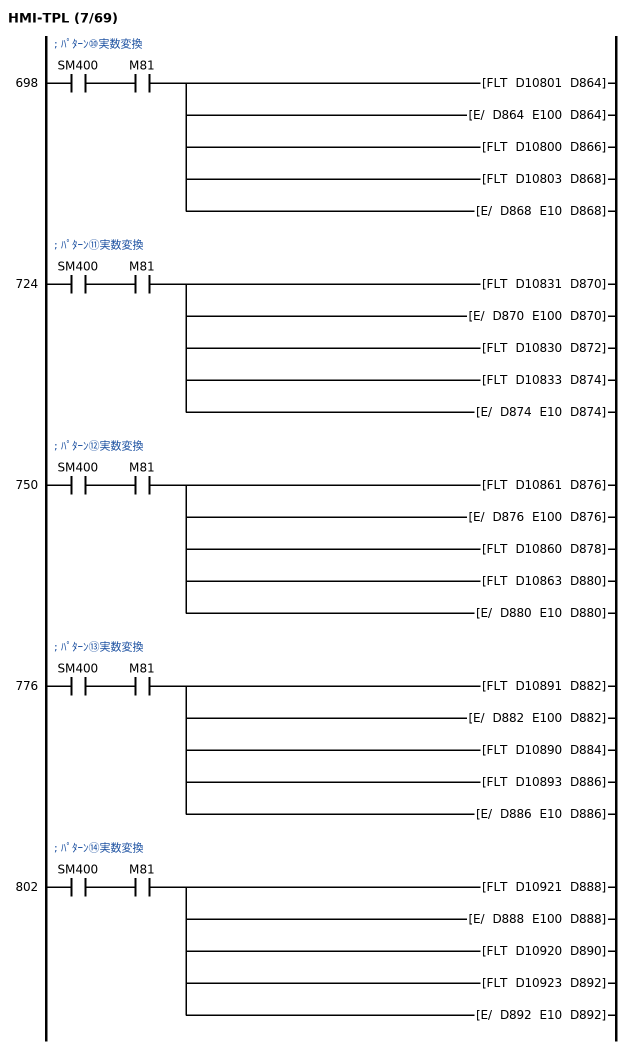
[picture p408: ladder of HMI-TPL, rungs at steps 698 to 802]
; ﾊﾟﾀｰﾝ⑩実数変換
698   LD      SM400
      AND     M81
      FLT     D10801 D864
      E/      D864 E100 D864
      FLT     D10800 D866
      FLT     D10803 D868
      E/      D868 E10 D868
; ﾊﾟﾀｰﾝ⑪実数変換
724   LD      SM400
      AND     M81
      FLT     D10831 D870
      E/      D870 E100 D870
      FLT     D10830 D872
      FLT     D10833 D874
      E/      D874 E10 D874
; ﾊﾟﾀｰﾝ⑫実数変換
750   LD      SM400
      AND     M81
      FLT     D10861 D876
      E/      D876 E100 D876
      FLT     D10860 D878
      FLT     D10863 D880
      E/      D880 E10 D880
; ﾊﾟﾀｰﾝ⑬実数変換
776   LD      SM400
      AND     M81
      FLT     D10891 D882
      E/      D882 E100 D882
      FLT     D10890 D884
      FLT     D10893 D886
      E/      D886 E10 D886
; ﾊﾟﾀｰﾝ⑭実数変換
802   LD      SM400
      AND     M81
      FLT     D10921 D888
      E/      D888 E100 D888
      FLT     D10920 D890
      FLT     D10923 D892
      E/      D892 E10 D892
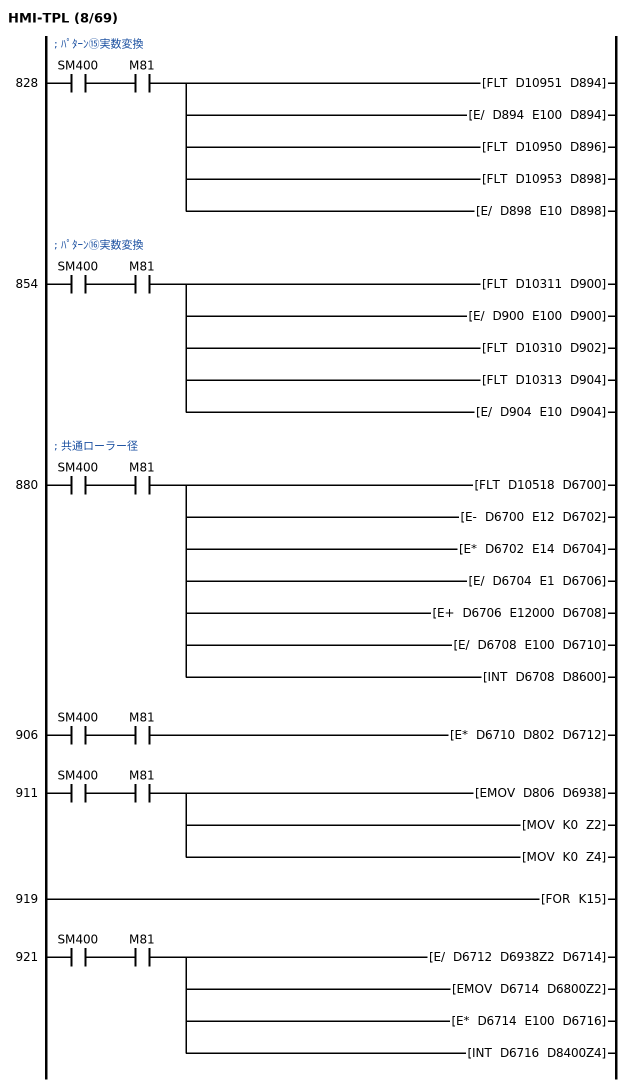
; ﾊﾟﾀｰﾝ⑮実数変換
828   LD      SM400
      AND     M81
      FLT     D10951 D894
      E/      D894 E100 D894
      FLT     D10950 D896
      FLT     D10953 D898
      E/      D898 E10 D898
; ﾊﾟﾀｰﾝ⑯実数変換
854   LD      SM400
      AND     M81
      FLT     D10311 D900
      E/      D900 E100 D900
      FLT     D10310 D902
      FLT     D10313 D904
      E/      D904 E10 D904
; 共通ローラー径
880   LD      SM400
      AND     M81
      FLT     D10518 D6700
      E-      D6700 E12 D6702
      E*      D6702 E14 D6704
      E/      D6704 E1 D6706
      E+      D6706 E12000 D6708
      E/      D6708 E100 D6710
      INT     D6708 D8600
906   LD      SM400
      AND     M81
      E*      D6710 D802 D6712
911   LD      SM400
      AND     M81
      EMOV    D806 D6938
      MOV     K0 Z2
      MOV     K0 Z4
919   FOR     K15
921   LD      SM400
      AND     M81
      E/      D6712 D6938Z2 D6714
      EMOV    D6714 D6800Z2
      E*      D6714 E100 D6716
      INT     D6716 D8400Z4
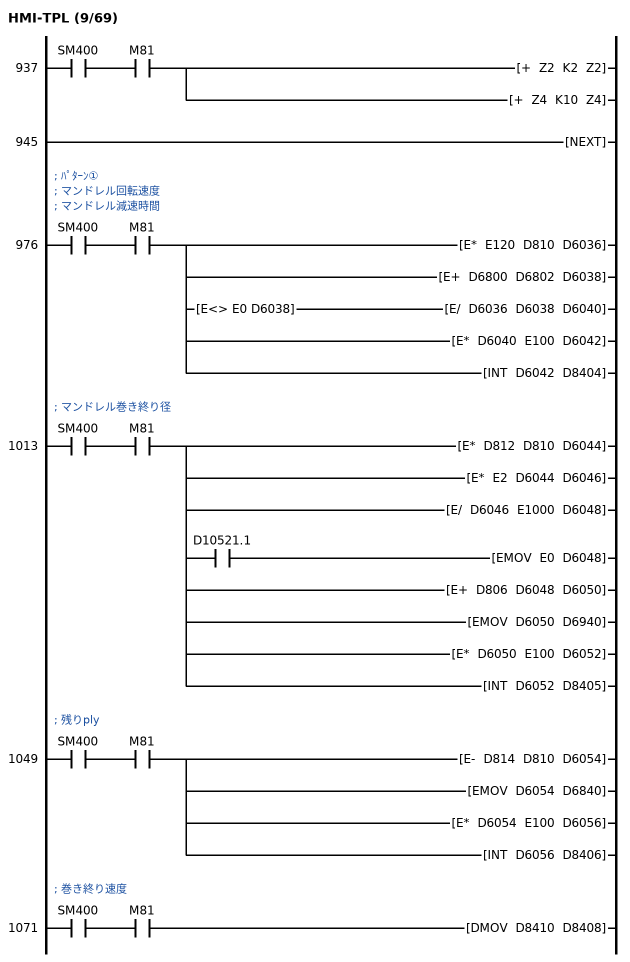
937   LD      SM400
      AND     M81
      +       Z2 K2 Z2
      +       Z4 K10 Z4
945   NEXT
; ﾊﾟﾀｰﾝ①
; マンドレル回転速度
; マンドレル減速時間
976   LD      SM400
      AND     M81
      E*      E120 D810 D6036
      E+      D6800 D6802 D6038
      MPS
      ANDE<>  E0 D6038
      E/      D6036 D6038 D6040
      MPP
      E*      D6040 E100 D6042
      INT     D6042 D8404
; マンドレル巻き終り径
1013  LD      SM400
      AND     M81
      E*      D812 D810 D6044
      E*      E2 D6044 D6046
      E/      D6046 E1000 D6048
      MPS
      AND     D10521.1
      EMOV    E0 D6048
      MPP
      E+      D806 D6048 D6050
      EMOV    D6050 D6940
      E*      D6050 E100 D6052
      INT     D6052 D8405
; 残りply
1049  LD      SM400
      AND     M81
      E-      D814 D810 D6054
      EMOV    D6054 D6840
      E*      D6054 E100 D6056
      INT     D6056 D8406
; 巻き終り速度
1071  LD      SM400
      AND     M81
      DMOV    D8410 D8408
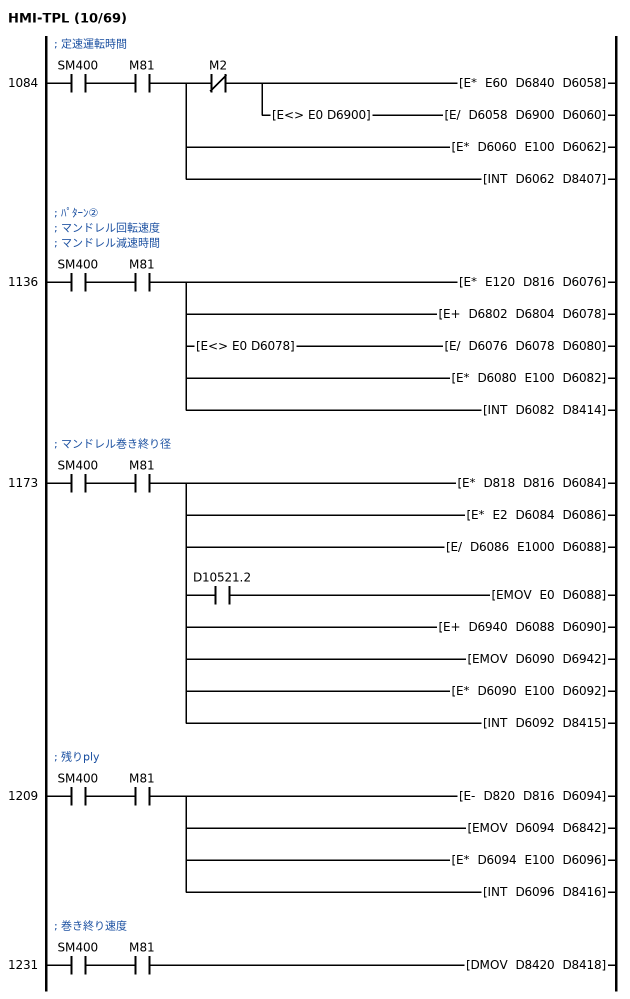
; 定速運転時間
1084  LD      SM400
      AND     M81
      MPS
      ANI     M2
      E*      E60 D6840 D6058
      ANDE<>  E0 D6900
      E/      D6058 D6900 D6060
      MPP
      E*      D6060 E100 D6062
      INT     D6062 D8407
; ﾊﾟﾀｰﾝ②
; マンドレル回転速度
; マンドレル減速時間
1136  LD      SM400
      AND     M81
      E*      E120 D816 D6076
      E+      D6802 D6804 D6078
      MPS
      ANDE<>  E0 D6078
      E/      D6076 D6078 D6080
      MPP
      E*      D6080 E100 D6082
      INT     D6082 D8414
; マンドレル巻き終り径
1173  LD      SM400
      AND     M81
      E*      D818 D816 D6084
      E*      E2 D6084 D6086
      E/      D6086 E1000 D6088
      MPS
      AND     D10521.2
      EMOV    E0 D6088
      MPP
      E+      D6940 D6088 D6090
      EMOV    D6090 D6942
      E*      D6090 E100 D6092
      INT     D6092 D8415
; 残りply
1209  LD      SM400
      AND     M81
      E-      D820 D816 D6094
      EMOV    D6094 D6842
      E*      D6094 E100 D6096
      INT     D6096 D8416
; 巻き終り速度
1231  LD      SM400
      AND     M81
      DMOV    D8420 D8418
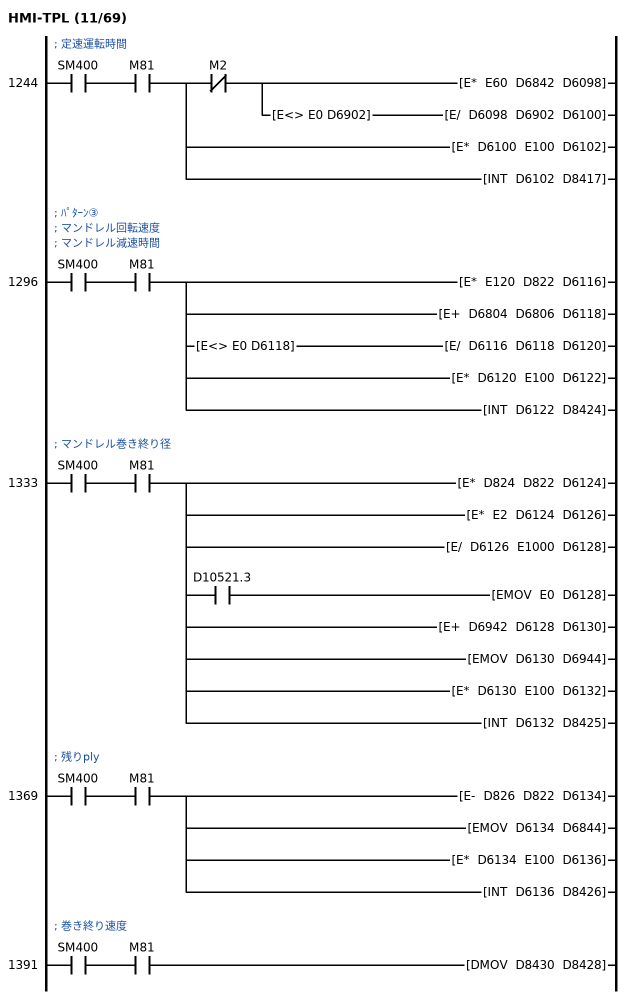
; 定速運転時間
1244  LD      SM400
      AND     M81
      MPS
      ANI     M2
      E*      E60 D6842 D6098
      ANDE<>  E0 D6902
      E/      D6098 D6902 D6100
      MPP
      E*      D6100 E100 D6102
      INT     D6102 D8417
; ﾊﾟﾀｰﾝ③
; マンドレル回転速度
; マンドレル減速時間
1296  LD      SM400
      AND     M81
      E*      E120 D822 D6116
      E+      D6804 D6806 D6118
      MPS
      ANDE<>  E0 D6118
      E/      D6116 D6118 D6120
      MPP
      E*      D6120 E100 D6122
      INT     D6122 D8424
; マンドレル巻き終り径
1333  LD      SM400
      AND     M81
      E*      D824 D822 D6124
      E*      E2 D6124 D6126
      E/      D6126 E1000 D6128
      MPS
      AND     D10521.3
      EMOV    E0 D6128
      MPP
      E+      D6942 D6128 D6130
      EMOV    D6130 D6944
      E*      D6130 E100 D6132
      INT     D6132 D8425
; 残りply
1369  LD      SM400
      AND     M81
      E-      D826 D822 D6134
      EMOV    D6134 D6844
      E*      D6134 E100 D6136
      INT     D6136 D8426
; 巻き終り速度
1391  LD      SM400
      AND     M81
      DMOV    D8430 D8428
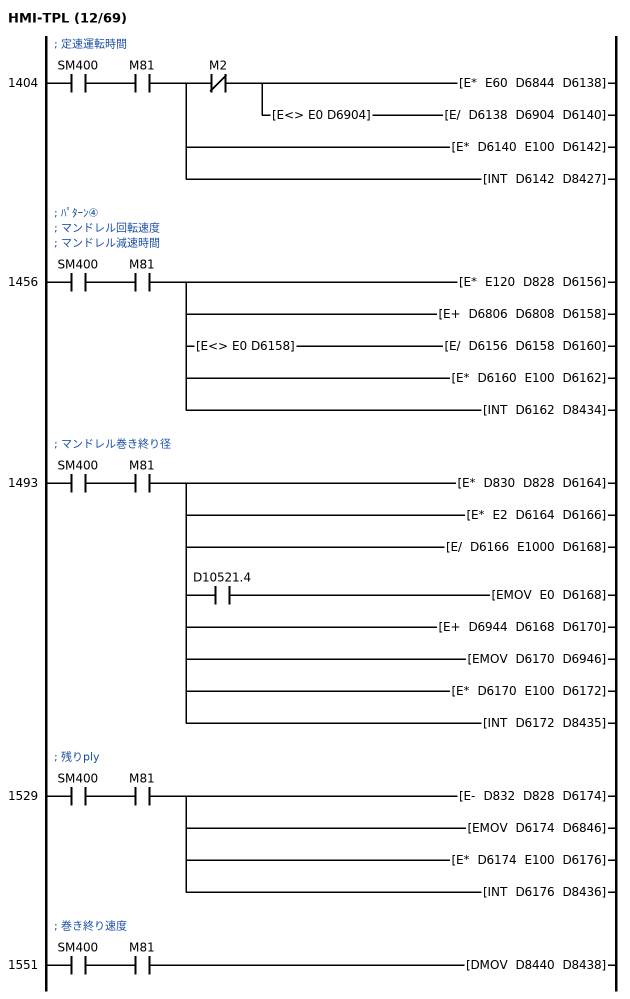
; 定速運転時間
1404  LD      SM400
      AND     M81
      MPS
      ANI     M2
      E*      E60 D6844 D6138
      ANDE<>  E0 D6904
      E/      D6138 D6904 D6140
      MPP
      E*      D6140 E100 D6142
      INT     D6142 D8427
; ﾊﾟﾀｰﾝ④
; マンドレル回転速度
; マンドレル減速時間
1456  LD      SM400
      AND     M81
      E*      E120 D828 D6156
      E+      D6806 D6808 D6158
      MPS
      ANDE<>  E0 D6158
      E/      D6156 D6158 D6160
      MPP
      E*      D6160 E100 D6162
      INT     D6162 D8434
; マンドレル巻き終り径
1493  LD      SM400
      AND     M81
      E*      D830 D828 D6164
      E*      E2 D6164 D6166
      E/      D6166 E1000 D6168
      MPS
      AND     D10521.4
      EMOV    E0 D6168
      MPP
      E+      D6944 D6168 D6170
      EMOV    D6170 D6946
      E*      D6170 E100 D6172
      INT     D6172 D8435
; 残りply
1529  LD      SM400
      AND     M81
      E-      D832 D828 D6174
      EMOV    D6174 D6846
      E*      D6174 E100 D6176
      INT     D6176 D8436
; 巻き終り速度
1551  LD      SM400
      AND     M81
      DMOV    D8440 D8438
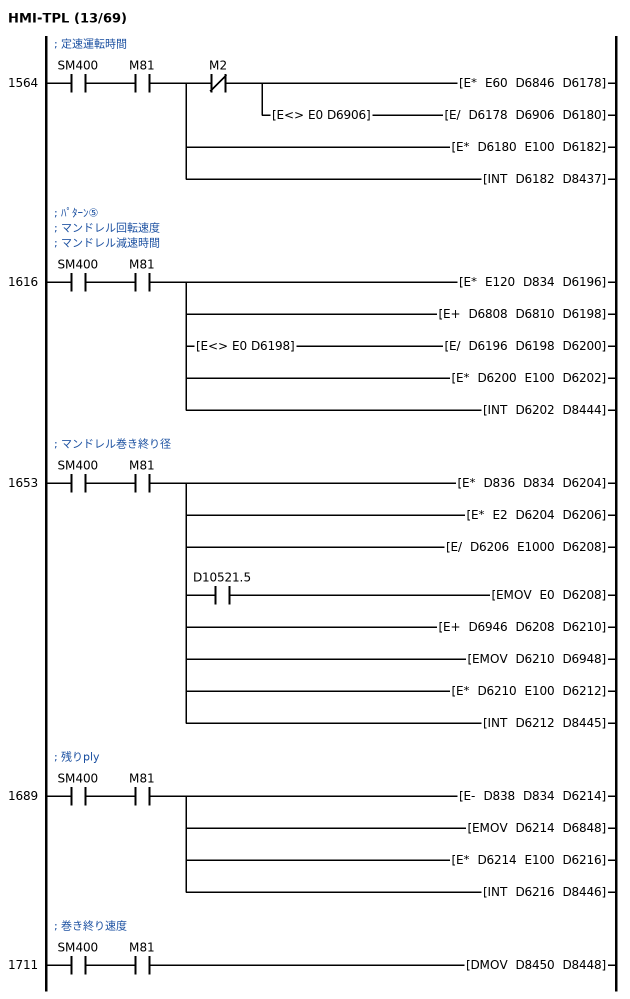
; 定速運転時間
1564  LD      SM400
      AND     M81
      MPS
      ANI     M2
      E*      E60 D6846 D6178
      ANDE<>  E0 D6906
      E/      D6178 D6906 D6180
      MPP
      E*      D6180 E100 D6182
      INT     D6182 D8437
; ﾊﾟﾀｰﾝ⑤
; マンドレル回転速度
; マンドレル減速時間
1616  LD      SM400
      AND     M81
      E*      E120 D834 D6196
      E+      D6808 D6810 D6198
      MPS
      ANDE<>  E0 D6198
      E/      D6196 D6198 D6200
      MPP
      E*      D6200 E100 D6202
      INT     D6202 D8444
; マンドレル巻き終り径
1653  LD      SM400
      AND     M81
      E*      D836 D834 D6204
      E*      E2 D6204 D6206
      E/      D6206 E1000 D6208
      MPS
      AND     D10521.5
      EMOV    E0 D6208
      MPP
      E+      D6946 D6208 D6210
      EMOV    D6210 D6948
      E*      D6210 E100 D6212
      INT     D6212 D8445
; 残りply
1689  LD      SM400
      AND     M81
      E-      D838 D834 D6214
      EMOV    D6214 D6848
      E*      D6214 E100 D6216
      INT     D6216 D8446
; 巻き終り速度
1711  LD      SM400
      AND     M81
      DMOV    D8450 D8448
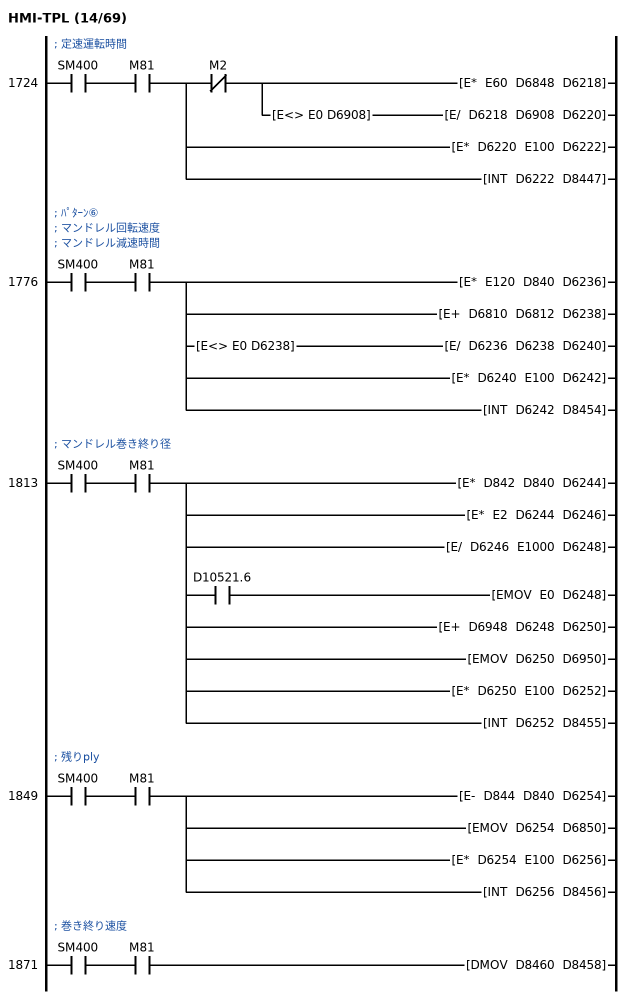
; 定速運転時間
1724  LD      SM400
      AND     M81
      MPS
      ANI     M2
      E*      E60 D6848 D6218
      ANDE<>  E0 D6908
      E/      D6218 D6908 D6220
      MPP
      E*      D6220 E100 D6222
      INT     D6222 D8447
; ﾊﾟﾀｰﾝ⑥
; マンドレル回転速度
; マンドレル減速時間
1776  LD      SM400
      AND     M81
      E*      E120 D840 D6236
      E+      D6810 D6812 D6238
      MPS
      ANDE<>  E0 D6238
      E/      D6236 D6238 D6240
      MPP
      E*      D6240 E100 D6242
      INT     D6242 D8454
; マンドレル巻き終り径
1813  LD      SM400
      AND     M81
      E*      D842 D840 D6244
      E*      E2 D6244 D6246
      E/      D6246 E1000 D6248
      MPS
      AND     D10521.6
      EMOV    E0 D6248
      MPP
      E+      D6948 D6248 D6250
      EMOV    D6250 D6950
      E*      D6250 E100 D6252
      INT     D6252 D8455
; 残りply
1849  LD      SM400
      AND     M81
      E-      D844 D840 D6254
      EMOV    D6254 D6850
      E*      D6254 E100 D6256
      INT     D6256 D8456
; 巻き終り速度
1871  LD      SM400
      AND     M81
      DMOV    D8460 D8458
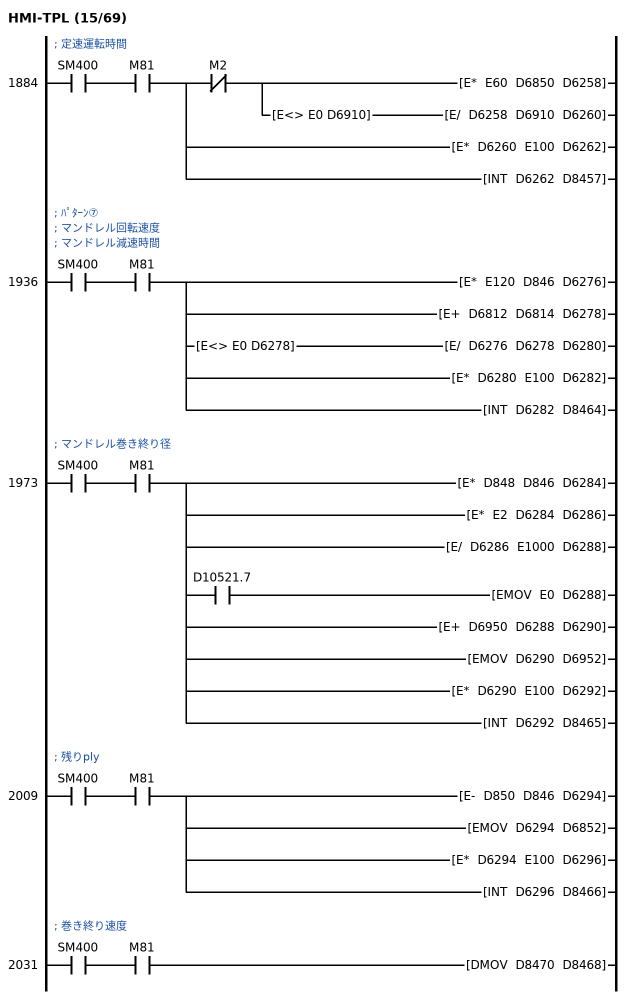
; 定速運転時間
1884  LD      SM400
      AND     M81
      MPS
      ANI     M2
      E*      E60 D6850 D6258
      ANDE<>  E0 D6910
      E/      D6258 D6910 D6260
      MPP
      E*      D6260 E100 D6262
      INT     D6262 D8457
; ﾊﾟﾀｰﾝ⑦
; マンドレル回転速度
; マンドレル減速時間
1936  LD      SM400
      AND     M81
      E*      E120 D846 D6276
      E+      D6812 D6814 D6278
      MPS
      ANDE<>  E0 D6278
      E/      D6276 D6278 D6280
      MPP
      E*      D6280 E100 D6282
      INT     D6282 D8464
; マンドレル巻き終り径
1973  LD      SM400
      AND     M81
      E*      D848 D846 D6284
      E*      E2 D6284 D6286
      E/      D6286 E1000 D6288
      MPS
      AND     D10521.7
      EMOV    E0 D6288
      MPP
      E+      D6950 D6288 D6290
      EMOV    D6290 D6952
      E*      D6290 E100 D6292
      INT     D6292 D8465
; 残りply
2009  LD      SM400
      AND     M81
      E-      D850 D846 D6294
      EMOV    D6294 D6852
      E*      D6294 E100 D6296
      INT     D6296 D8466
; 巻き終り速度
2031  LD      SM400
      AND     M81
      DMOV    D8470 D8468
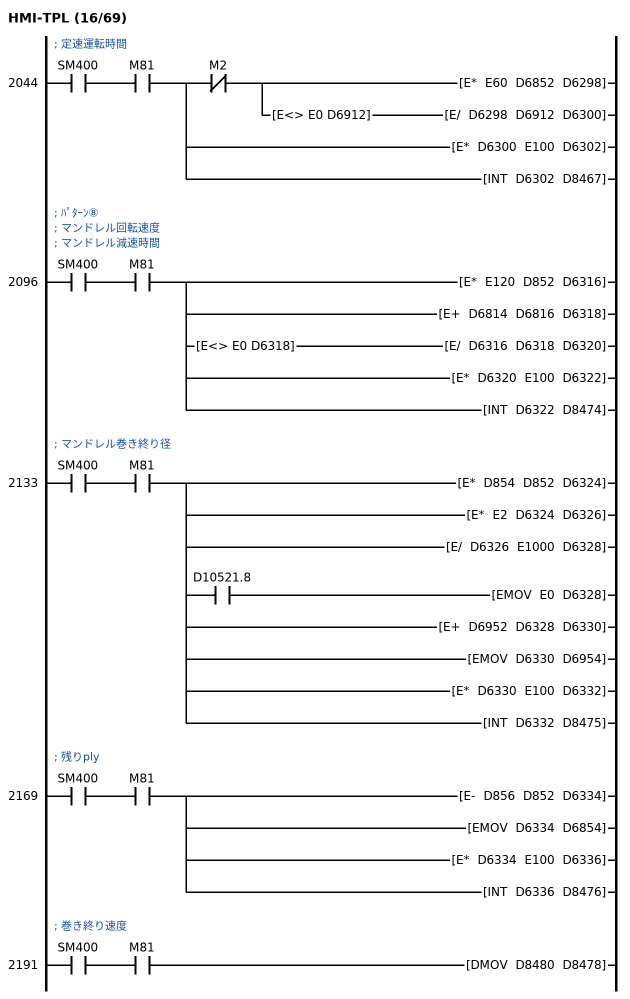
; 定速運転時間
2044  LD      SM400
      AND     M81
      MPS
      ANI     M2
      E*      E60 D6852 D6298
      ANDE<>  E0 D6912
      E/      D6298 D6912 D6300
      MPP
      E*      D6300 E100 D6302
      INT     D6302 D8467
; ﾊﾟﾀｰﾝ⑧
; マンドレル回転速度
; マンドレル減速時間
2096  LD      SM400
      AND     M81
      E*      E120 D852 D6316
      E+      D6814 D6816 D6318
      MPS
      ANDE<>  E0 D6318
      E/      D6316 D6318 D6320
      MPP
      E*      D6320 E100 D6322
      INT     D6322 D8474
; マンドレル巻き終り径
2133  LD      SM400
      AND     M81
      E*      D854 D852 D6324
      E*      E2 D6324 D6326
      E/      D6326 E1000 D6328
      MPS
      AND     D10521.8
      EMOV    E0 D6328
      MPP
      E+      D6952 D6328 D6330
      EMOV    D6330 D6954
      E*      D6330 E100 D6332
      INT     D6332 D8475
; 残りply
2169  LD      SM400
      AND     M81
      E-      D856 D852 D6334
      EMOV    D6334 D6854
      E*      D6334 E100 D6336
      INT     D6336 D8476
; 巻き終り速度
2191  LD      SM400
      AND     M81
      DMOV    D8480 D8478
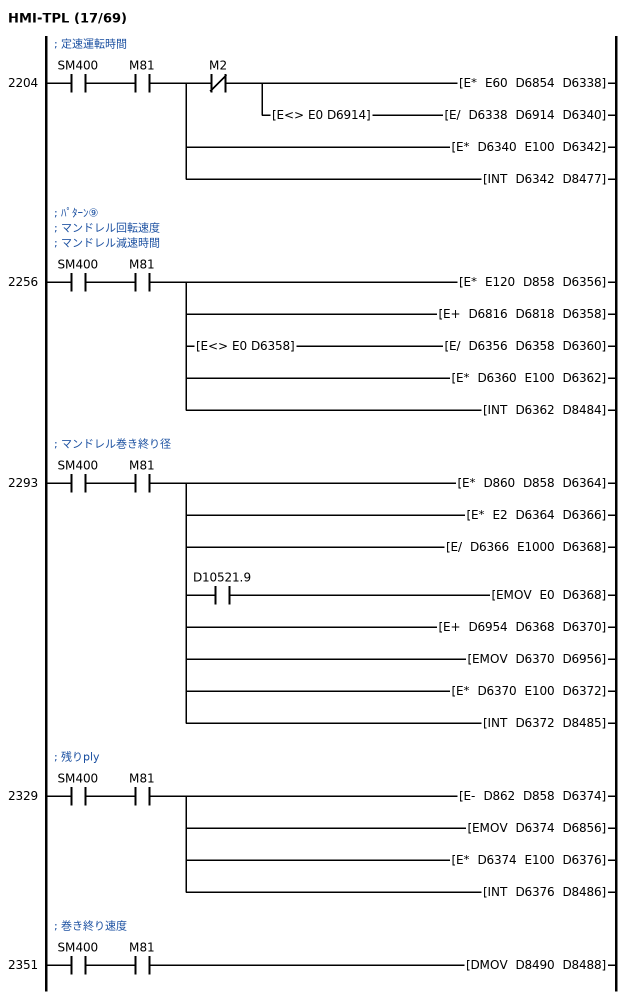
; 定速運転時間
2204  LD      SM400
      AND     M81
      MPS
      ANI     M2
      E*      E60 D6854 D6338
      ANDE<>  E0 D6914
      E/      D6338 D6914 D6340
      MPP
      E*      D6340 E100 D6342
      INT     D6342 D8477
; ﾊﾟﾀｰﾝ⑨
; マンドレル回転速度
; マンドレル減速時間
2256  LD      SM400
      AND     M81
      E*      E120 D858 D6356
      E+      D6816 D6818 D6358
      MPS
      ANDE<>  E0 D6358
      E/      D6356 D6358 D6360
      MPP
      E*      D6360 E100 D6362
      INT     D6362 D8484
; マンドレル巻き終り径
2293  LD      SM400
      AND     M81
      E*      D860 D858 D6364
      E*      E2 D6364 D6366
      E/      D6366 E1000 D6368
      MPS
      AND     D10521.9
      EMOV    E0 D6368
      MPP
      E+      D6954 D6368 D6370
      EMOV    D6370 D6956
      E*      D6370 E100 D6372
      INT     D6372 D8485
; 残りply
2329  LD      SM400
      AND     M81
      E-      D862 D858 D6374
      EMOV    D6374 D6856
      E*      D6374 E100 D6376
      INT     D6376 D8486
; 巻き終り速度
2351  LD      SM400
      AND     M81
      DMOV    D8490 D8488
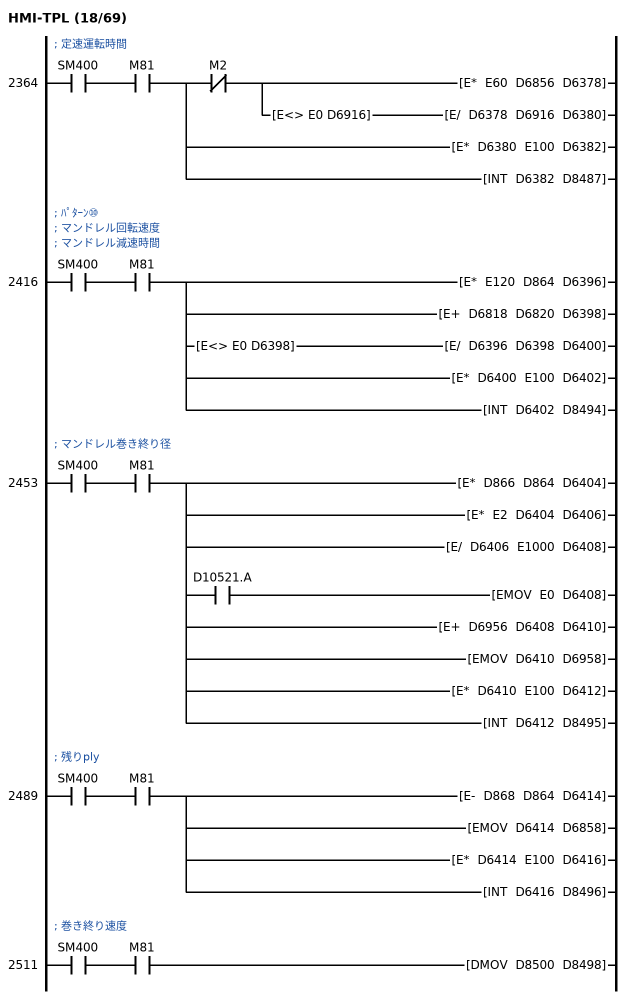
; 定速運転時間
2364  LD      SM400
      AND     M81
      MPS
      ANI     M2
      E*      E60 D6856 D6378
      ANDE<>  E0 D6916
      E/      D6378 D6916 D6380
      MPP
      E*      D6380 E100 D6382
      INT     D6382 D8487
; ﾊﾟﾀｰﾝ⑩
; マンドレル回転速度
; マンドレル減速時間
2416  LD      SM400
      AND     M81
      E*      E120 D864 D6396
      E+      D6818 D6820 D6398
      MPS
      ANDE<>  E0 D6398
      E/      D6396 D6398 D6400
      MPP
      E*      D6400 E100 D6402
      INT     D6402 D8494
; マンドレル巻き終り径
2453  LD      SM400
      AND     M81
      E*      D866 D864 D6404
      E*      E2 D6404 D6406
      E/      D6406 E1000 D6408
      MPS
      AND     D10521.A
      EMOV    E0 D6408
      MPP
      E+      D6956 D6408 D6410
      EMOV    D6410 D6958
      E*      D6410 E100 D6412
      INT     D6412 D8495
; 残りply
2489  LD      SM400
      AND     M81
      E-      D868 D864 D6414
      EMOV    D6414 D6858
      E*      D6414 E100 D6416
      INT     D6416 D8496
; 巻き終り速度
2511  LD      SM400
      AND     M81
      DMOV    D8500 D8498
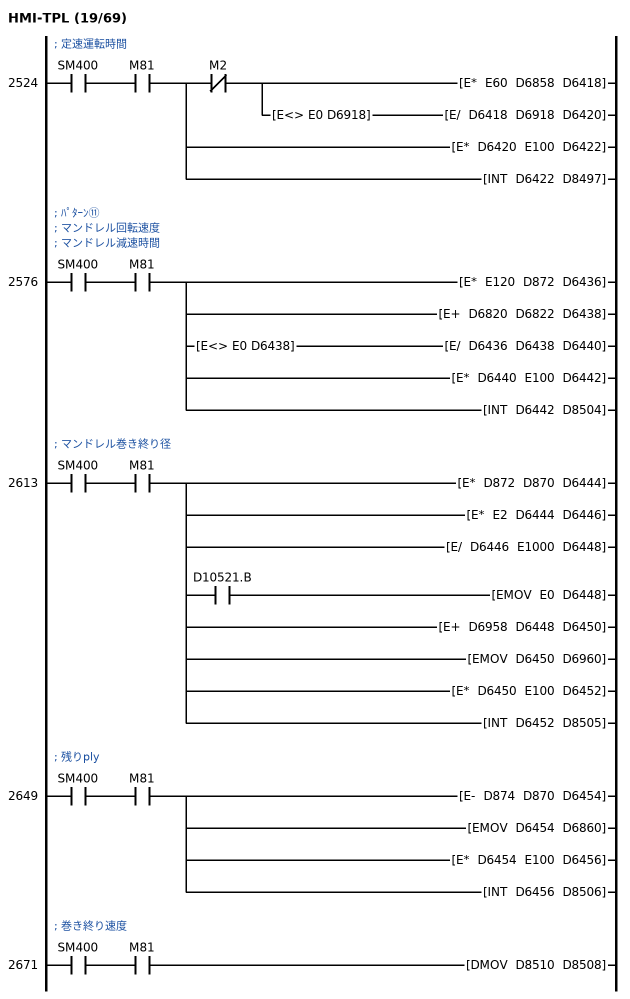
; 定速運転時間
2524  LD      SM400
      AND     M81
      MPS
      ANI     M2
      E*      E60 D6858 D6418
      ANDE<>  E0 D6918
      E/      D6418 D6918 D6420
      MPP
      E*      D6420 E100 D6422
      INT     D6422 D8497
; ﾊﾟﾀｰﾝ⑪
; マンドレル回転速度
; マンドレル減速時間
2576  LD      SM400
      AND     M81
      E*      E120 D872 D6436
      E+      D6820 D6822 D6438
      MPS
      ANDE<>  E0 D6438
      E/      D6436 D6438 D6440
      MPP
      E*      D6440 E100 D6442
      INT     D6442 D8504
; マンドレル巻き終り径
2613  LD      SM400
      AND     M81
      E*      D872 D870 D6444
      E*      E2 D6444 D6446
      E/      D6446 E1000 D6448
      MPS
      AND     D10521.B
      EMOV    E0 D6448
      MPP
      E+      D6958 D6448 D6450
      EMOV    D6450 D6960
      E*      D6450 E100 D6452
      INT     D6452 D8505
; 残りply
2649  LD      SM400
      AND     M81
      E-      D874 D870 D6454
      EMOV    D6454 D6860
      E*      D6454 E100 D6456
      INT     D6456 D8506
; 巻き終り速度
2671  LD      SM400
      AND     M81
      DMOV    D8510 D8508
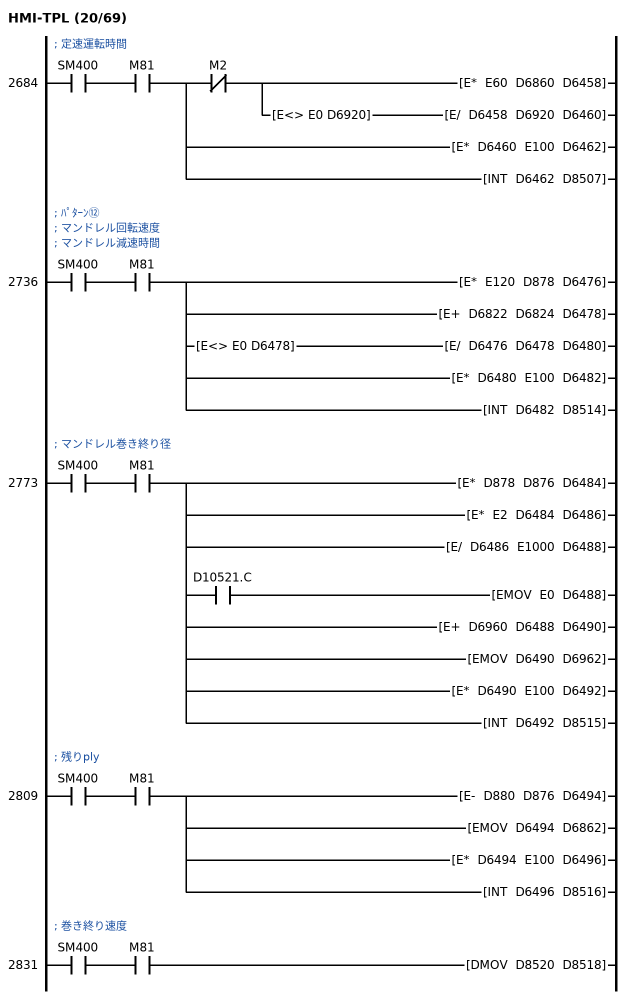
; 定速運転時間
2684  LD      SM400
      AND     M81
      MPS
      ANI     M2
      E*      E60 D6860 D6458
      ANDE<>  E0 D6920
      E/      D6458 D6920 D6460
      MPP
      E*      D6460 E100 D6462
      INT     D6462 D8507
; ﾊﾟﾀｰﾝ⑫
; マンドレル回転速度
; マンドレル減速時間
2736  LD      SM400
      AND     M81
      E*      E120 D878 D6476
      E+      D6822 D6824 D6478
      MPS
      ANDE<>  E0 D6478
      E/      D6476 D6478 D6480
      MPP
      E*      D6480 E100 D6482
      INT     D6482 D8514
; マンドレル巻き終り径
2773  LD      SM400
      AND     M81
      E*      D878 D876 D6484
      E*      E2 D6484 D6486
      E/      D6486 E1000 D6488
      MPS
      AND     D10521.C
      EMOV    E0 D6488
      MPP
      E+      D6960 D6488 D6490
      EMOV    D6490 D6962
      E*      D6490 E100 D6492
      INT     D6492 D8515
; 残りply
2809  LD      SM400
      AND     M81
      E-      D880 D876 D6494
      EMOV    D6494 D6862
      E*      D6494 E100 D6496
      INT     D6496 D8516
; 巻き終り速度
2831  LD      SM400
      AND     M81
      DMOV    D8520 D8518
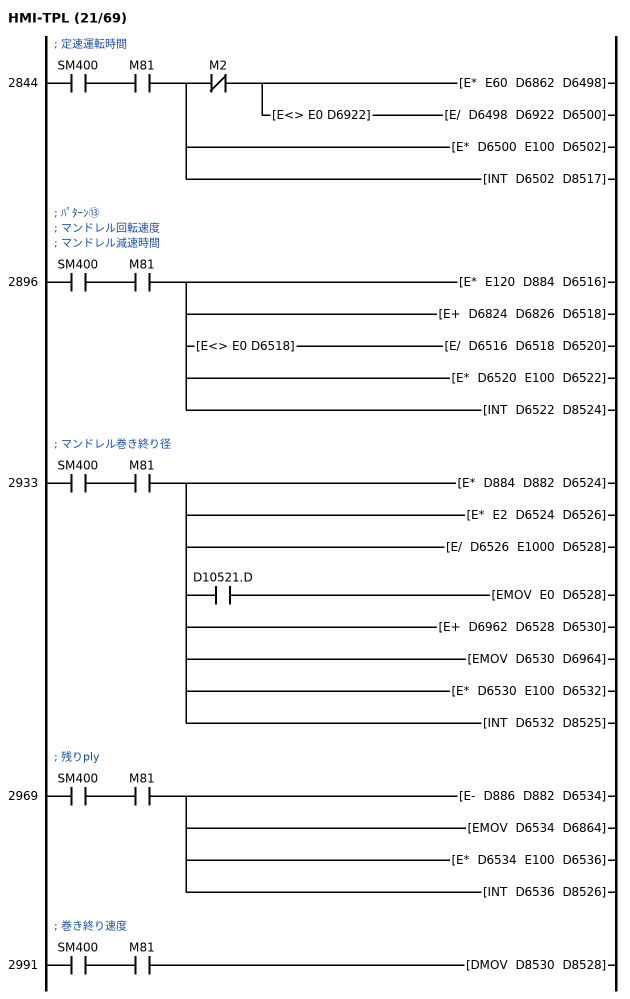
; 定速運転時間
2844  LD      SM400
      AND     M81
      MPS
      ANI     M2
      E*      E60 D6862 D6498
      ANDE<>  E0 D6922
      E/      D6498 D6922 D6500
      MPP
      E*      D6500 E100 D6502
      INT     D6502 D8517
; ﾊﾟﾀｰﾝ⑬
; マンドレル回転速度
; マンドレル減速時間
2896  LD      SM400
      AND     M81
      E*      E120 D884 D6516
      E+      D6824 D6826 D6518
      MPS
      ANDE<>  E0 D6518
      E/      D6516 D6518 D6520
      MPP
      E*      D6520 E100 D6522
      INT     D6522 D8524
; マンドレル巻き終り径
2933  LD      SM400
      AND     M81
      E*      D884 D882 D6524
      E*      E2 D6524 D6526
      E/      D6526 E1000 D6528
      MPS
      AND     D10521.D
      EMOV    E0 D6528
      MPP
      E+      D6962 D6528 D6530
      EMOV    D6530 D6964
      E*      D6530 E100 D6532
      INT     D6532 D8525
; 残りply
2969  LD      SM400
      AND     M81
      E-      D886 D882 D6534
      EMOV    D6534 D6864
      E*      D6534 E100 D6536
      INT     D6536 D8526
; 巻き終り速度
2991  LD      SM400
      AND     M81
      DMOV    D8530 D8528
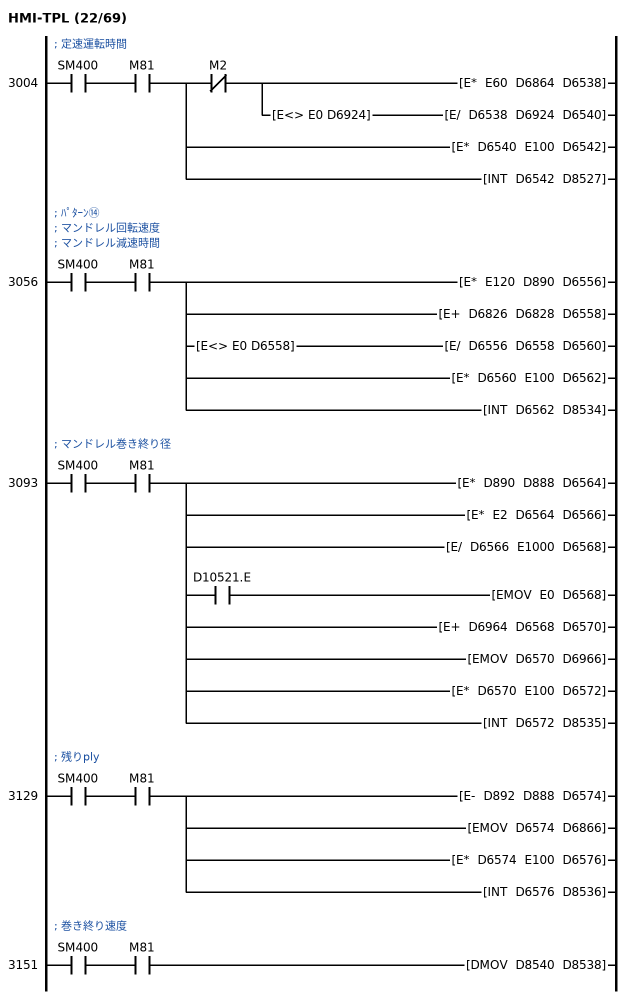
; 定速運転時間
3004  LD      SM400
      AND     M81
      MPS
      ANI     M2
      E*      E60 D6864 D6538
      ANDE<>  E0 D6924
      E/      D6538 D6924 D6540
      MPP
      E*      D6540 E100 D6542
      INT     D6542 D8527
; ﾊﾟﾀｰﾝ⑭
; マンドレル回転速度
; マンドレル減速時間
3056  LD      SM400
      AND     M81
      E*      E120 D890 D6556
      E+      D6826 D6828 D6558
      MPS
      ANDE<>  E0 D6558
      E/      D6556 D6558 D6560
      MPP
      E*      D6560 E100 D6562
      INT     D6562 D8534
; マンドレル巻き終り径
3093  LD      SM400
      AND     M81
      E*      D890 D888 D6564
      E*      E2 D6564 D6566
      E/      D6566 E1000 D6568
      MPS
      AND     D10521.E
      EMOV    E0 D6568
      MPP
      E+      D6964 D6568 D6570
      EMOV    D6570 D6966
      E*      D6570 E100 D6572
      INT     D6572 D8535
; 残りply
3129  LD      SM400
      AND     M81
      E-      D892 D888 D6574
      EMOV    D6574 D6866
      E*      D6574 E100 D6576
      INT     D6576 D8536
; 巻き終り速度
3151  LD      SM400
      AND     M81
      DMOV    D8540 D8538
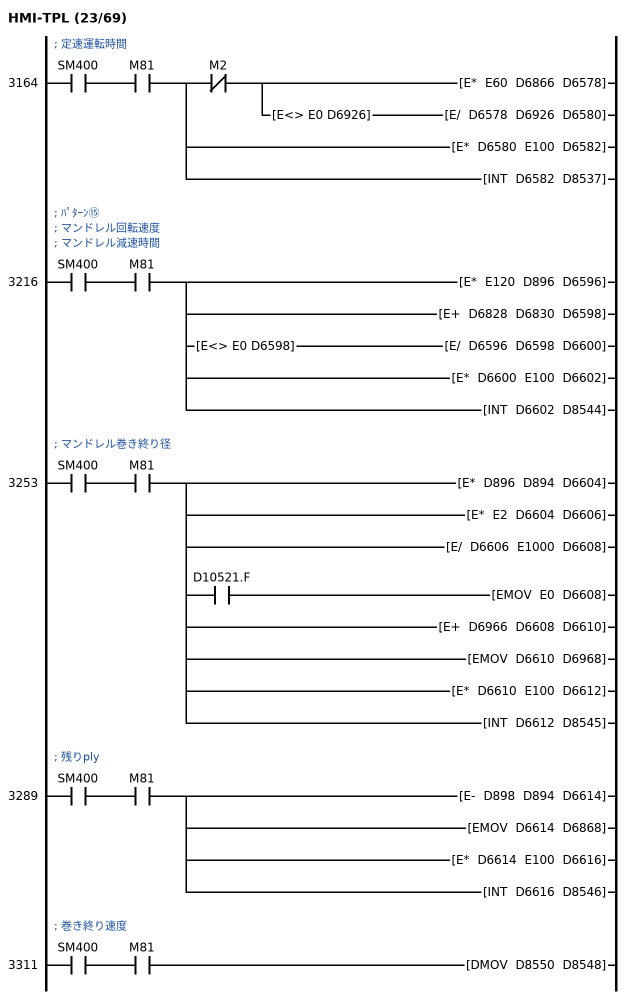
; 定速運転時間
3164  LD      SM400
      AND     M81
      MPS
      ANI     M2
      E*      E60 D6866 D6578
      ANDE<>  E0 D6926
      E/      D6578 D6926 D6580
      MPP
      E*      D6580 E100 D6582
      INT     D6582 D8537
; ﾊﾟﾀｰﾝ⑮
; マンドレル回転速度
; マンドレル減速時間
3216  LD      SM400
      AND     M81
      E*      E120 D896 D6596
      E+      D6828 D6830 D6598
      MPS
      ANDE<>  E0 D6598
      E/      D6596 D6598 D6600
      MPP
      E*      D6600 E100 D6602
      INT     D6602 D8544
; マンドレル巻き終り径
3253  LD      SM400
      AND     M81
      E*      D896 D894 D6604
      E*      E2 D6604 D6606
      E/      D6606 E1000 D6608
      MPS
      AND     D10521.F
      EMOV    E0 D6608
      MPP
      E+      D6966 D6608 D6610
      EMOV    D6610 D6968
      E*      D6610 E100 D6612
      INT     D6612 D8545
; 残りply
3289  LD      SM400
      AND     M81
      E-      D898 D894 D6614
      EMOV    D6614 D6868
      E*      D6614 E100 D6616
      INT     D6616 D8546
; 巻き終り速度
3311  LD      SM400
      AND     M81
      DMOV    D8550 D8548
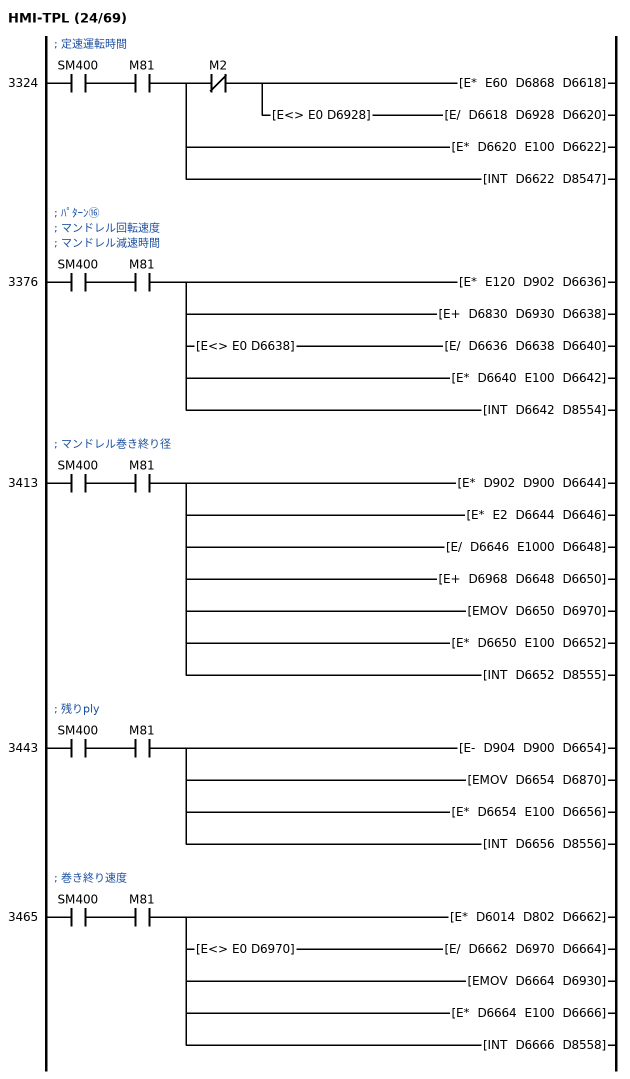
; 定速運転時間
3324  LD      SM400
      AND     M81
      MPS
      ANI     M2
      E*      E60 D6868 D6618
      ANDE<>  E0 D6928
      E/      D6618 D6928 D6620
      MPP
      E*      D6620 E100 D6622
      INT     D6622 D8547
; ﾊﾟﾀｰﾝ⑯
; マンドレル回転速度
; マンドレル減速時間
3376  LD      SM400
      AND     M81
      E*      E120 D902 D6636
      E+      D6830 D6930 D6638
      MPS
      ANDE<>  E0 D6638
      E/      D6636 D6638 D6640
      MPP
      E*      D6640 E100 D6642
      INT     D6642 D8554
; マンドレル巻き終り径
3413  LD      SM400
      AND     M81
      E*      D902 D900 D6644
      E*      E2 D6644 D6646
      E/      D6646 E1000 D6648
      E+      D6968 D6648 D6650
      EMOV    D6650 D6970
      E*      D6650 E100 D6652
      INT     D6652 D8555
; 残りply
3443  LD      SM400
      AND     M81
      E-      D904 D900 D6654
      EMOV    D6654 D6870
      E*      D6654 E100 D6656
      INT     D6656 D8556
; 巻き終り速度
3465  LD      SM400
      AND     M81
      E*      D6014 D802 D6662
      MPS
      ANDE<>  E0 D6970
      E/      D6662 D6970 D6664
      MPP
      EMOV    D6664 D6930
      E*      D6664 E100 D6666
      INT     D6666 D8558
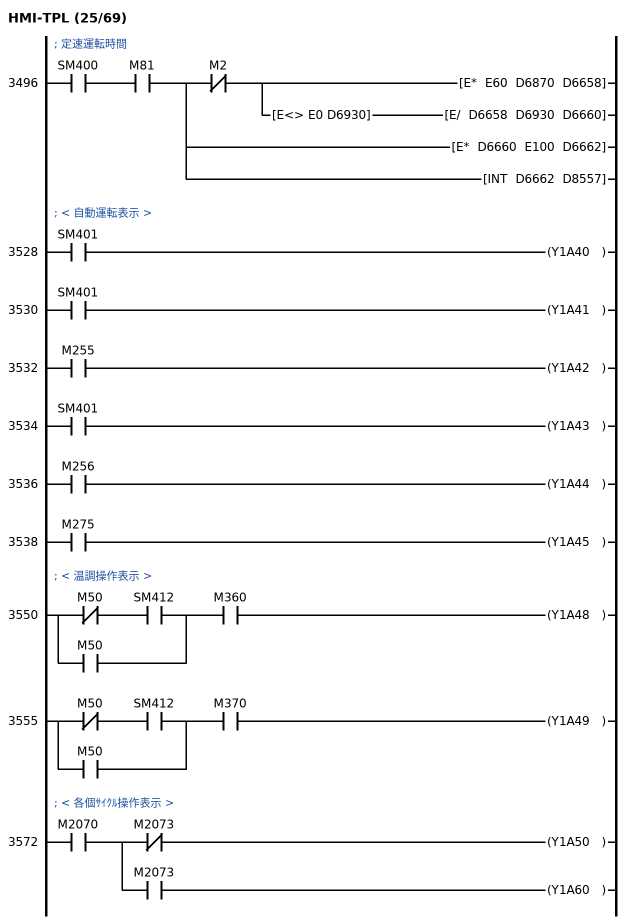
; 定速運転時間
3496  LD      SM400
      AND     M81
      MPS
      ANI     M2
      E*      E60 D6870 D6658
      ANDE<>  E0 D6930
      E/      D6658 D6930 D6660
      MPP
      E*      D6660 E100 D6662
      INT     D6662 D8557
; < 自動運転表示 >
3528  LD      SM401
      OUT     Y1A40
3530  LD      SM401
      OUT     Y1A41
3532  LD      M255
      OUT     Y1A42
3534  LD      SM401
      OUT     Y1A43
3536  LD      M256
      OUT     Y1A44
3538  LD      M275
      OUT     Y1A45
; < 温調操作表示 >
3550  LDI     M50
      AND     SM412
      OR      M50
      AND     M360
      OUT     Y1A48
3555  LDI     M50
      AND     SM412
      OR      M50
      AND     M370
      OUT     Y1A49
; < 各個ｻｲｸﾙ操作表示 >
3572  LD      M2070
      MPS
      ANI     M2073
      OUT     Y1A50
      MPP
      AND     M2073
      OUT     Y1A60
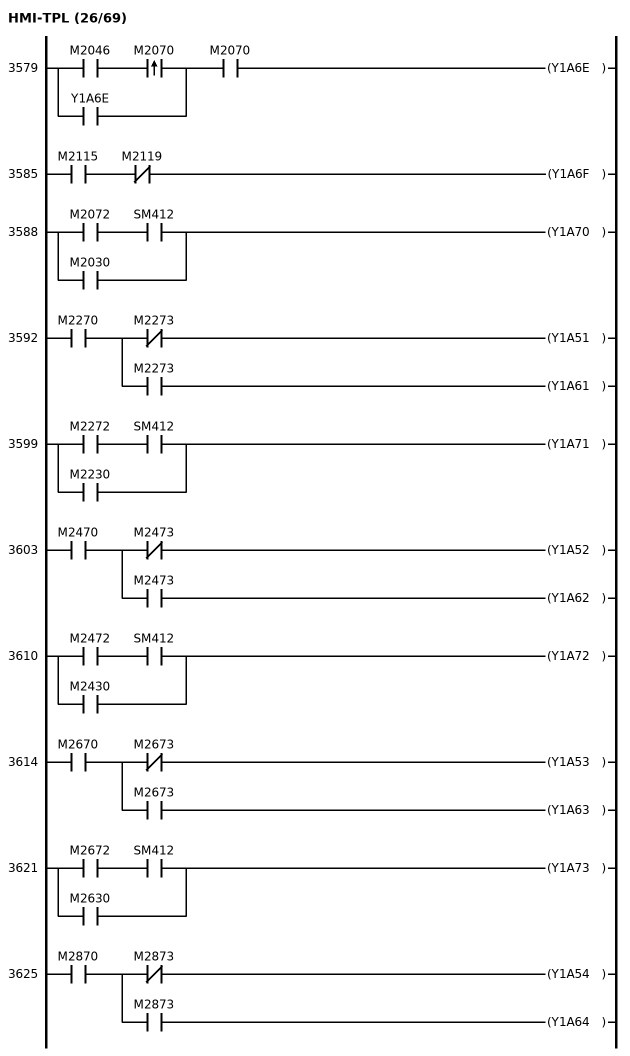
3579  LD      M2046
      ANDP    M2070
      OR      Y1A6E
      AND     M2070
      OUT     Y1A6E
3585  LD      M2115
      ANI     M2119
      OUT     Y1A6F
3588  LD      M2072
      AND     SM412
      OR      M2030
      OUT     Y1A70
3592  LD      M2270
      MPS
      ANI     M2273
      OUT     Y1A51
      MPP
      AND     M2273
      OUT     Y1A61
3599  LD      M2272
      AND     SM412
      OR      M2230
      OUT     Y1A71
3603  LD      M2470
      MPS
      ANI     M2473
      OUT     Y1A52
      MPP
      AND     M2473
      OUT     Y1A62
3610  LD      M2472
      AND     SM412
      OR      M2430
      OUT     Y1A72
3614  LD      M2670
      MPS
      ANI     M2673
      OUT     Y1A53
      MPP
      AND     M2673
      OUT     Y1A63
3621  LD      M2672
      AND     SM412
      OR      M2630
      OUT     Y1A73
3625  LD      M2870
      MPS
      ANI     M2873
      OUT     Y1A54
      MPP
      AND     M2873
      OUT     Y1A64
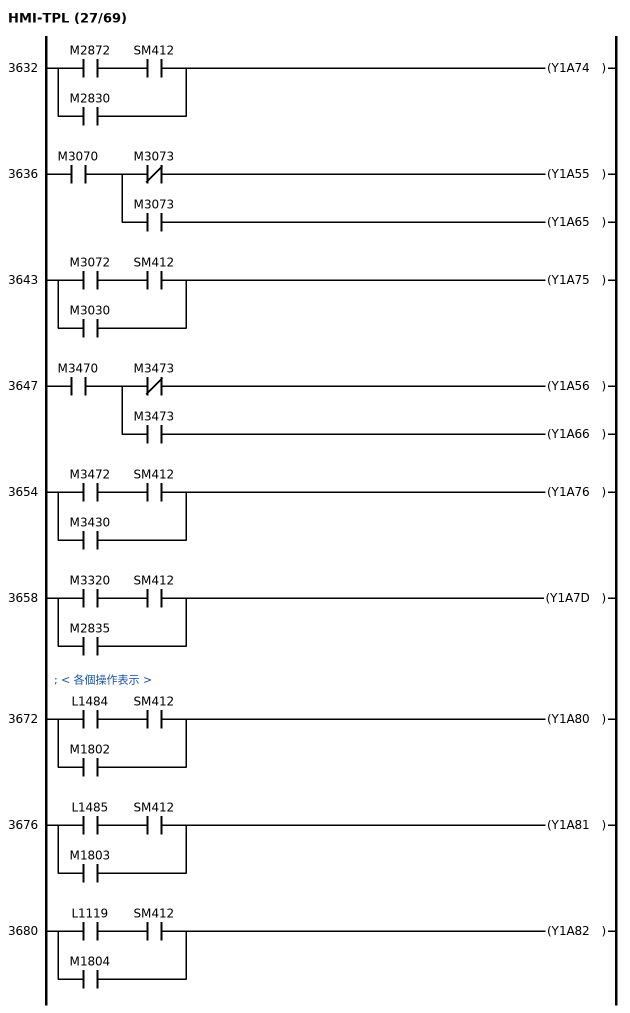
3632  LD      M2872
      AND     SM412
      OR      M2830
      OUT     Y1A74
3636  LD      M3070
      MPS
      ANI     M3073
      OUT     Y1A55
      MPP
      AND     M3073
      OUT     Y1A65
3643  LD      M3072
      AND     SM412
      OR      M3030
      OUT     Y1A75
3647  LD      M3470
      MPS
      ANI     M3473
      OUT     Y1A56
      MPP
      AND     M3473
      OUT     Y1A66
3654  LD      M3472
      AND     SM412
      OR      M3430
      OUT     Y1A76
3658  LD      M3320
      AND     SM412
      OR      M2835
      OUT     Y1A7D
; < 各個操作表示 >
3672  LD      L1484
      AND     SM412
      OR      M1802
      OUT     Y1A80
3676  LD      L1485
      AND     SM412
      OR      M1803
      OUT     Y1A81
3680  LD      L1119
      AND     SM412
      OR      M1804
      OUT     Y1A82
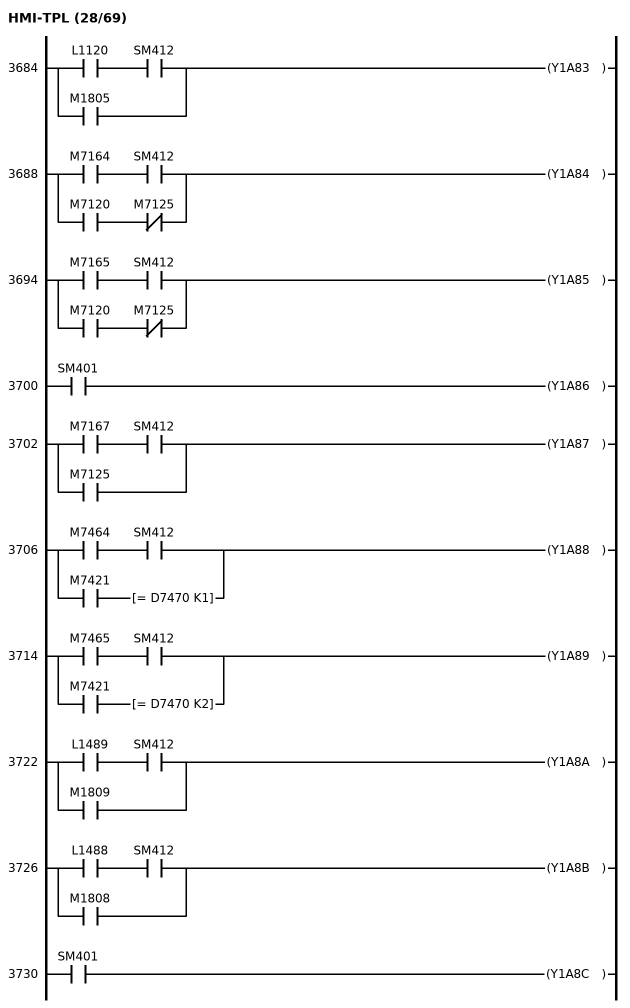
3684  LD      L1120
      AND     SM412
      OR      M1805
      OUT     Y1A83
3688  LD      M7164
      AND     SM412
      LD      M7120
      ANI     M7125
      ORB
      OUT     Y1A84
3694  LD      M7165
      AND     SM412
      LD      M7120
      ANI     M7125
      ORB
      OUT     Y1A85
3700  LD      SM401
      OUT     Y1A86
3702  LD      M7167
      AND     SM412
      OR      M7125
      OUT     Y1A87
3706  LD      M7464
      AND     SM412
      LD      M7421
      AND=    D7470 K1
      ORB
      OUT     Y1A88
3714  LD      M7465
      AND     SM412
      LD      M7421
      AND=    D7470 K2
      ORB
      OUT     Y1A89
3722  LD      L1489
      AND     SM412
      OR      M1809
      OUT     Y1A8A
3726  LD      L1488
      AND     SM412
      OR      M1808
      OUT     Y1A8B
3730  LD      SM401
      OUT     Y1A8C
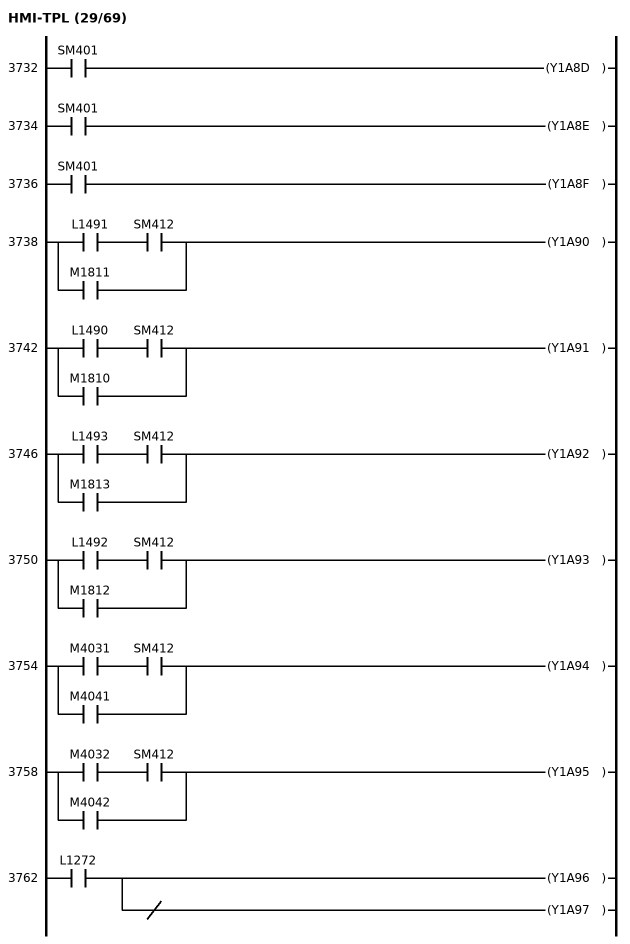
3732  LD      SM401
      OUT     Y1A8D
3734  LD      SM401
      OUT     Y1A8E
3736  LD      SM401
      OUT     Y1A8F
3738  LD      L1491
      AND     SM412
      OR      M1811
      OUT     Y1A90
3742  LD      L1490
      AND     SM412
      OR      M1810
      OUT     Y1A91
3746  LD      L1493
      AND     SM412
      OR      M1813
      OUT     Y1A92
3750  LD      L1492
      AND     SM412
      OR      M1812
      OUT     Y1A93
3754  LD      M4031
      AND     SM412
      OR      M4041
      OUT     Y1A94
3758  LD      M4032
      AND     SM412
      OR      M4042
      OUT     Y1A95
3762  LD      L1272
      OUT     Y1A96
      INV
      OUT     Y1A97
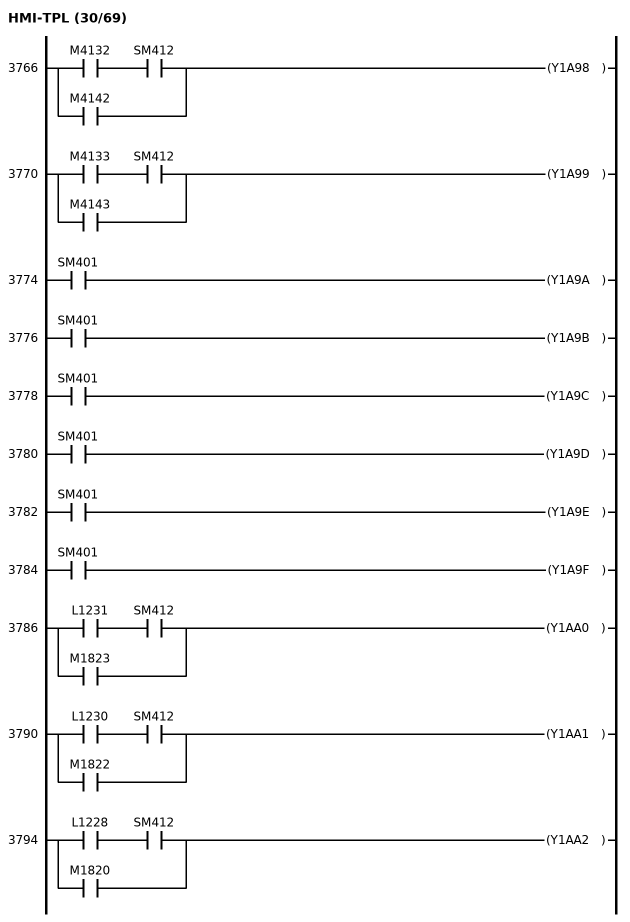
3766  LD      M4132
      AND     SM412
      OR      M4142
      OUT     Y1A98
3770  LD      M4133
      AND     SM412
      OR      M4143
      OUT     Y1A99
3774  LD      SM401
      OUT     Y1A9A
3776  LD      SM401
      OUT     Y1A9B
3778  LD      SM401
      OUT     Y1A9C
3780  LD      SM401
      OUT     Y1A9D
3782  LD      SM401
      OUT     Y1A9E
3784  LD      SM401
      OUT     Y1A9F
3786  LD      L1231
      AND     SM412
      OR      M1823
      OUT     Y1AA0
3790  LD      L1230
      AND     SM412
      OR      M1822
      OUT     Y1AA1
3794  LD      L1228
      AND     SM412
      OR      M1820
      OUT     Y1AA2
